// TIA Portal V20 export
DATA_BLOCK "Instance_FB_Send_Water_Fountain_To_Rework_DB"   // DB108
// stored: AutoNumber false, InstanceOfName FB_Send_Water_Fountain_To_Rework, InstanceOfType FB
"FB_Send_Water_Fountain_To_Rework"
   // VAR_INPUT
   //    Emergency_Stop_Release : Bool;
   //    Start : Bool;
   //    Water_Fountain_Fail_Test : Bool;
   //    Trigger_Read_Serial_Number_Exit_Functional_Test : Bool;
   //    Sensor_Water_Fountain_Exit_Functional_Test_Spinner_Conveyor_Belt : Bool;
   //    Sensor_Spinner_Exit_Functional_Test_Position_Withdrawn : Bool;
   //    Sensor_Spinner_Exit_Functional_Test_Position_Advanced : Bool;
   //    Sensor_Water_Fountain_Exit_Functional_Test_After_Spinner_Conveyor_Belt : Bool;
   //    Sensor_Water_Fountain_Geting_Entrace_Rework_Conveyor_Belt_Start : Bool;
   // END_VAR
   // VAR_OUTPUT
   //    Turn_On_Conveyor_Belt_Motor_Spinner_Get_Exit_Functional_Test : Bool;
   //    Valve_Advance_Spinner_Get_Exit_Functional_Test : Bool;
   //    Pause_Conveyor_Belt_And_Carousel_Functional_Test : Bool;
   // END_VAR
   // VAR
   //    Aux_Trig_0 : Bool;
   //    Aux_Trig_1 : Bool;
   //    Aux_Trig_2 : Bool;
   //    Aux_Trig_3 : Bool;
   //    Aux_Trig_4 : Bool;
   //    Aux_Trig_5 : Bool;
   //    Aux_Trig_6 : Bool;
   //    Aux_Trig_7 : Bool;
   //    Wait_Clean_Spinner : Bool;
   //    Wait_Get_In_Spinner : Bool;
   //    "Counter" : USInt;
   //    Timer_Delay_Turn_On_Motor_Spinner_Conveyor_Belt { S7_SetPoint := 'True'} : TON_TIME;
   // END_VAR
   // VAR RETAIN
   //    Counter_Water_Fountain_Exiting_Functional_Test { S7_SetPoint := 'True'} : CTUD_USINT;
   // END_VAR
BEGIN
END_DATA_BLOCK
